Omron CX-Programmer project NewProject (CX-Programmer 9.75)

# PLC NewPLC1: CP2E-N N

## Global symbols (name address type ; comment)
0.00 BOOL  ; PROXY STOP KONVEYOR
0.01 BOOL  ; PROXY BOWL DISPENSER 1
0.02 BOOL  ; START BUTTON
0.03 BOOL  ; PROXY BOWL DISPENSER 2
100.00 BOOL  ; MOTOR BOWL DISPENSER
100.01 BOOL  ; MOTOR KONVEYOR 1
100.02 BOOL  ; MOTOR KONVEYOR
100.06 BOOL  ; MOTOR LINEAR ACTUATOR
10.02 BOOL  ; Cup Dispensed
200.00 BOOL  ; RELAY START
200.01 BOOL  ; RELAY START KONVEYOR
200.02 BOOL  ; RELAY ACTUATOR
200.03 BOOL  ; MOTOR BOWL
200.04 BOOL  ; RESET COUNTER
C0 CHANNEL  ; COMPILE MOTOR BOWL
C000 BOOL  ; DispensingOrder Done
T000 BOOL  ; TIMER ActuatorMie
T001 BOOL  ; Timer Reset
T002 BOOL  ; TIMER START KONVEYOR AFTER BOWL
T003 BOOL  ; START BOWL
W100.01 BOOL  ; MieKering_Ready
W100.02 BOOL  ; Cup_Jalan
W100.03 BOOL  ; RebusMie1_Start
W100.04 BOOL  ; RebusMie1_Done
W100.05 BOOL  ; RebusMie2_Start
W100.06 BOOL  ; RebusMie2_Done
W100.07 BOOL  ; RebusMie3_Start
W100.08 BOOL  ; RebusMie3_Done
W100.09 BOOL  ; Picked Cup
W10.00 BOOL  ; RST
W10.01 BOOL  ; MieKering_Picked
W10.02 BOOL  ; Cup dispensed
W10.03 BOOL  ; CupReady
W11.00 BOOL  ; Delay 1sec Trigger
W12.00 BOOL  ; 1 Sec Delay
W1.00 BOOL  ; MieKering_Arrived
W1.01 BOOL  ; MieKering_Picked
W1.02 BOOL  ; Cup_Dropped
W2.00 BOOL  ; ModbusStatus
W2.01 BOOL  ; TIMRST
W2.02 BOOL  ; 1stOrder Done
W3.00 BOOL  ; StartRelay
W3.01 BOOL  ; MotorMie
W3.02 BOOL  ; Conveyor
W3.03 BOOL  ; Mie Sampe
W3.05 BOOL  ; BowlJatuh
W3.06 BOOL  ; Bowl Arrived
W3.07 BOOL  ; Second Cup
W5.00 BOOL  ; Start MODBUS
FB_MODBUSTCP_SERVER _CP2E003_ExecuteModTcpServer
Order1_Menu D110 CHANNEL
Order1_Topping1 D100 CHANNEL
Order1_Topping2 D101 CHANNEL
Order1_Topping3 D102 CHANNEL
Order2_Menu D111 CHANNEL
Order2_Topping1 D103 CHANNEL
Order2_Topping2 D104 CHANNEL
Order2_Topping3 D105 CHANNEL
Order3_Menu D112 CHANNEL
Order3_Topping1 D106 CHANNEL
Order3_Topping2 D107 CHANNEL
Order3_Topping3 D108 CHANNEL
Start_Order W100.00 BOOL

## Program MODBUS (cyclic task 0)

### Section MODBUS

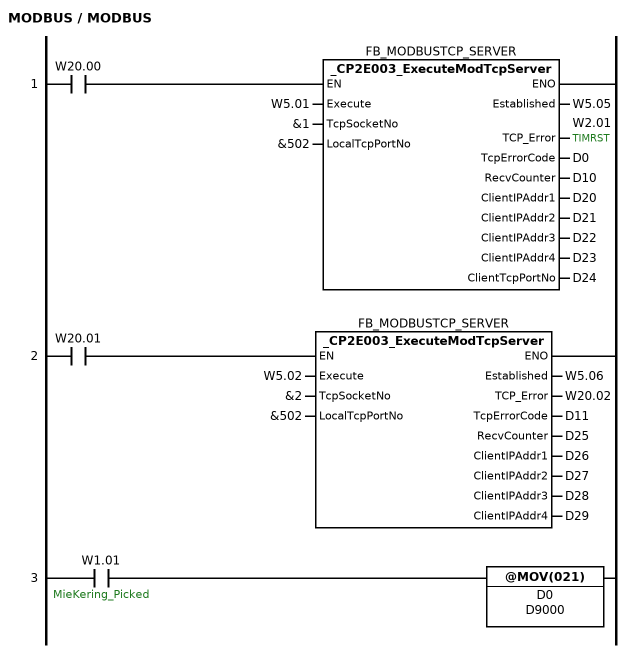
; rung 1
LD W20.00
CALL FB_MODBUSTCP_SERVER : _CP2E003_ExecuteModTcpServer (Execute := W5.01, TcpSocketNo := &1, LocalTcpPortNo := &502, Established => W5.05, TCP_Error => W2.01, TcpErrorCode => D0, RecvCounter => D10, ClientIPAddr1 => D20, ClientIPAddr2 => D21, ClientIPAddr3 => D22, ClientIPAddr4 => D23, ClientTcpPortNo => D24)  ; TIMRST
; rung 2
LD W20.01
CALL FB_MODBUSTCP_SERVER : _CP2E003_ExecuteModTcpServer (Execute := W5.02, TcpSocketNo := &2, LocalTcpPortNo := &502, Established => W5.06, TCP_Error => W20.02, TcpErrorCode => D11, RecvCounter => D25, ClientIPAddr1 => D26, ClientIPAddr2 => D27, ClientIPAddr3 => D28, ClientIPAddr4 => D29)
; rung 3
LD W1.01  ; MieKering_Picked
@MOV(021) D0 D9000

### Section Feeder_Main

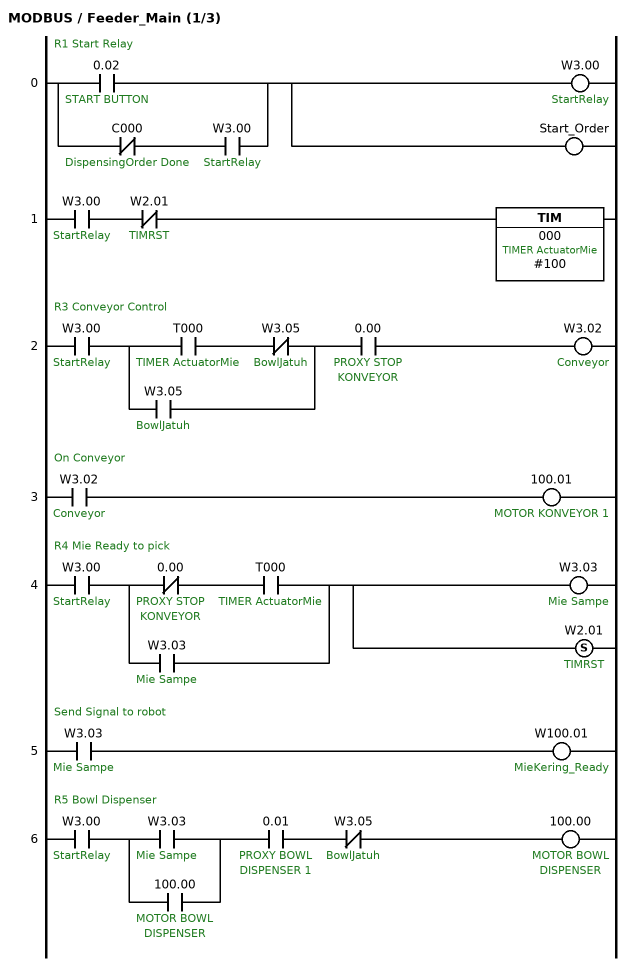
; rung 0: R1 Start Relay
LD 0.02  ; START BUTTON
LDNOT C000  ; DispensingOrder Done
AND W3.00  ; StartRelay
ORLD
OUT W3.00  ; StartRelay
OUT Start_Order
; rung 1
LD W3.00  ; StartRelay
ANDNOT W2.01  ; TIMRST
TIM 000 #100  ; TIMER ActuatorMie
; rung 2: R3 Conveyor Control
LD W3.00  ; StartRelay
LD T000  ; TIMER ActuatorMie
ANDNOT W3.05  ; BowlJatuh
OR W3.05  ; BowlJatuh
ANDLD
AND 0.00  ; PROXY STOP KONVEYOR
OUT W3.02  ; Conveyor
; rung 3: On Conveyor
LD W3.02  ; Conveyor
OUT 100.01  ; MOTOR KONVEYOR 1
; rung 4: R4 Mie Ready to pick
LD W3.00  ; StartRelay
LDNOT 0.00  ; PROXY STOP KONVEYOR
AND T000  ; TIMER ActuatorMie
OR W3.03  ; Mie Sampe
ANDLD
OUT W3.03  ; Mie Sampe
SET W2.01  ; TIMRST
; rung 5: Send Signal to robot
LD W3.03  ; Mie Sampe
OUT W100.01  ; MieKering_Ready
; rung 6: R5 Bowl Dispenser
LD W3.00  ; StartRelay
LD W3.03  ; Mie Sampe
OR 100.00  ; MOTOR BOWL DISPENSER
ANDLD
AND 0.01  ; PROXY BOWL DISPENSER 1
ANDNOT W3.05  ; BowlJatuh
OUT 100.00  ; MOTOR BOWL DISPENSER

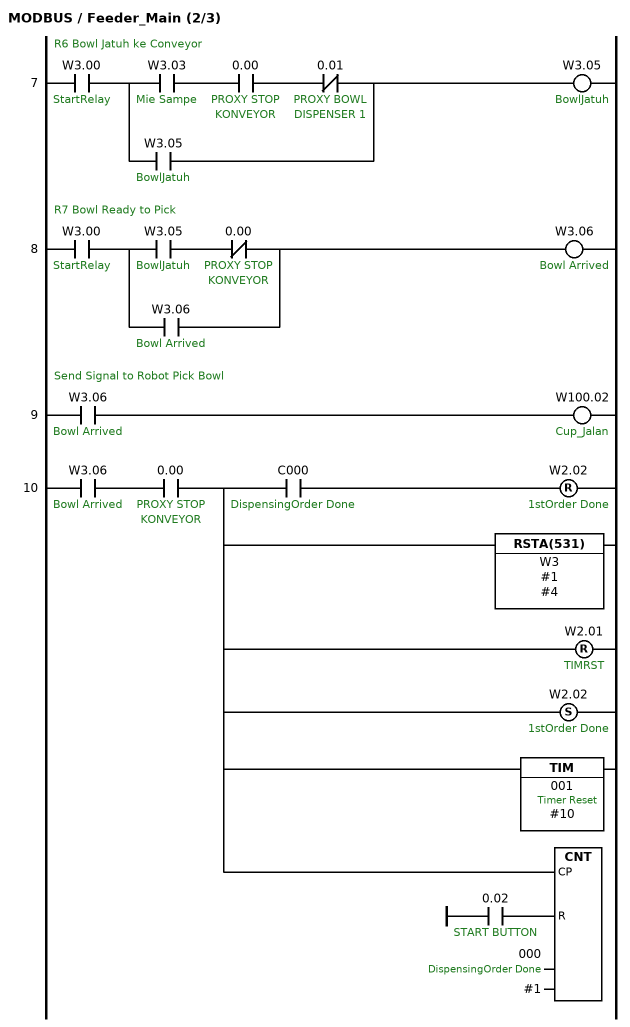
; rung 7: R6 Bowl Jatuh ke Conveyor
LD W3.00  ; StartRelay
LD W3.03  ; Mie Sampe
AND 0.00  ; PROXY STOP KONVEYOR
ANDNOT 0.01  ; PROXY BOWL DISPENSER 1
OR W3.05  ; BowlJatuh
ANDLD
OUT W3.05  ; BowlJatuh
; rung 8: R7 Bowl Ready to Pick
LD W3.00  ; StartRelay
LD W3.05  ; BowlJatuh
ANDNOT 0.00  ; PROXY STOP KONVEYOR
OR W3.06  ; Bowl Arrived
ANDLD
OUT W3.06  ; Bowl Arrived
; rung 9: Send Signal to Robot Pick Bowl
LD W3.06  ; Bowl Arrived
OUT W100.02  ; Cup_Jalan
; rung 10
LD W3.06  ; Bowl Arrived
AND 0.00  ; PROXY STOP KONVEYOR
OUT TR0
AND C000  ; DispensingOrder Done
RSET W2.02  ; 1stOrder Done
LD TR0
RSTA(531) W3 #1 #4
RSET W2.01  ; TIMRST
SET W2.02  ; 1stOrder Done
TIM 001 #10  ; Timer Reset
LD 0.02  ; START BUTTON
CNT 000 #1  ; DispensingOrder Done

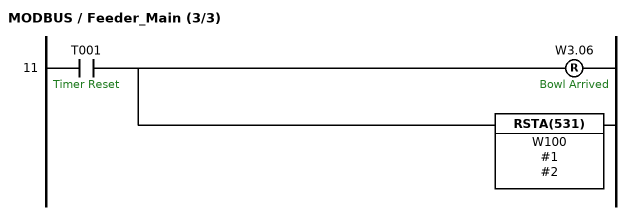
; rung 11
LD T001  ; Timer Reset
RSET W3.06  ; Bowl Arrived
RSTA(531) W100 #1 #2

### Section Delay_Timer

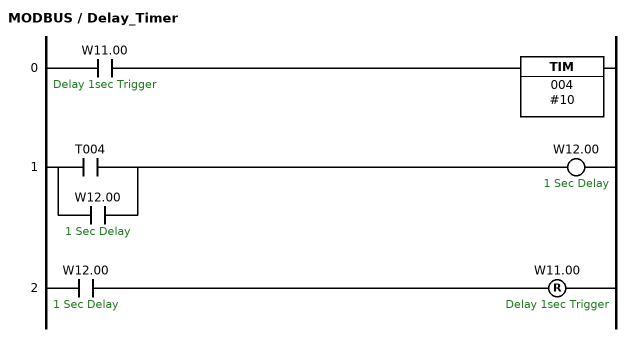
; rung 0
LD W11.00  ; Delay 1sec Trigger
TIM 004 #10
; rung 1
LD T004
OR W12.00  ; 1 Sec Delay
OUT W12.00  ; 1 Sec Delay
; rung 2
LD W12.00  ; 1 Sec Delay
RSET W11.00  ; Delay 1sec Trigger

### Section Feeder_MultiOrder

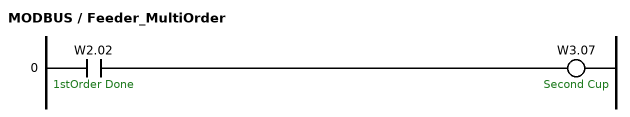
; rung 0
LD W2.02  ; 1stOrder Done
OUT W3.07  ; Second Cup

### Section Mie_Dispenser

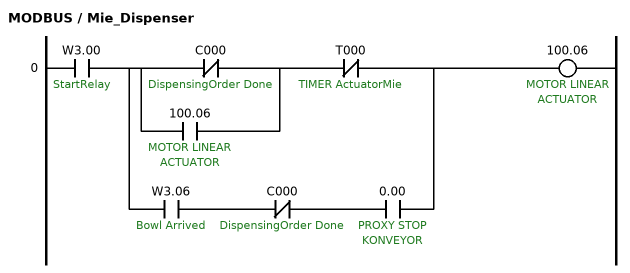
; rung 0
LD W3.00  ; StartRelay
LDNOT C000  ; DispensingOrder Done
OR 100.06  ; MOTOR LINEAR ACTUATOR
ANDNOT T000  ; TIMER ActuatorMie
LD W3.06  ; Bowl Arrived
ANDNOT C000  ; DispensingOrder Done
AND 0.00  ; PROXY STOP KONVEYOR
ORLD
ANDLD
OUT 100.06  ; MOTOR LINEAR ACTUATOR

### Section END
; rung 0
END(001)

## Function block _CP2E003_ExecuteModTcpServer (Omron library block, body left out)